FUNCTION_BLOCK FB_LT_REAL (* REAL Comparison *)
  (* Standard: 61499-1-D.1; Classification: Math *)
  (* Version 0.1, 2007-09-06, JHC, Holobloc Inc, Moved to fb.rt.compare. *)
  (* Version 0.0, 2002-03-11, JHC, Rockwell Automation *)
  (* Compiler header: package fb.rt.compare; *)
  (* Compiler classdef: public class FB_LT_REAL extends FB_GT_REAL *)
  (* Compiler Java Sun JDK 1.6.0 *)
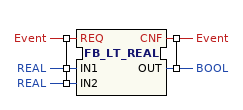
  EVENT_INPUT
    REQ WITH IN1, IN2;
  END_EVENT
  EVENT_OUTPUT
    CNF WITH OUT;
  END_EVENT
  VAR_INPUT
    IN1 : REAL;
    IN2 : REAL;
  END_VAR
  VAR_OUTPUT
    OUT : BOOL; (* IN1<IN2 *)
  END_VAR
END_FUNCTION_BLOCK
